{attribute 'qualified_only'}
{attribute 'strict'}
TYPE cPuckStatusEval :
(
	
	None := 0

) DINT;
END_TYPE

(* stored: Version 1.1.0.1, ProductVersion 3.1.4024.6
   DUT cPuckStatusEval: Id {35167b6d-587d-463e-a8b0-1a6474e2c386} *)
